ABB RobotStudio station: test1_20190225-122105.rsstn

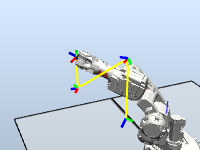
Station test1 (saved by RobotStudio 6.8.8148.134)
Layout (positions relative to the parent item):
  - IRB140_6_81_C_03_2 [mechanism, from Robots\IRB140_6_81_C_G_03.rslib] at (0, 0, 0) mm; joint values [-0.7275, 0.7441, -1.0821, -1.1758, 0.2324, 2.3516] (rad or m)
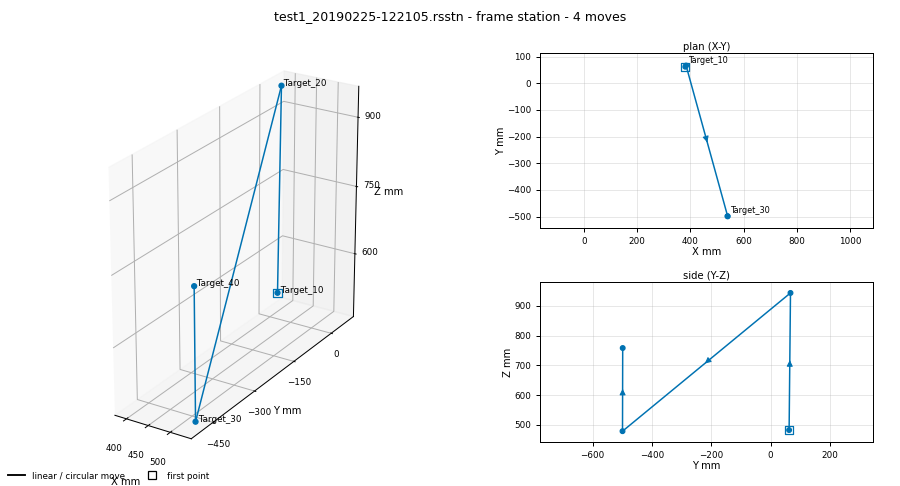
[picture p0: tool path of test1_20190225-122105.rsstn in frame station, 4 of 4 moves have a stored position in this frame; points joined in program order, loops and branches not executed]
Targets, tools, work objects and paths stored in the station, written as RAPID:
! task (no controller)
MODULE Module1
  CONST robtarget Target_10:=[[380.698967065,62.135252828,482.100752166],[0.23292276,-0.432299751,0.867192227,-0.082713687],[0,-1,-1,0],[9E+09,9E+09,9E+09,9E+09,9E+09,9E+09]];
  CONST robtarget Target_20:=[[383.520804221,66.771067435,943.970503399],[0.810617732,-0.21605232,0.523687989,-0.148226777],[0,0,-1,0],[9E+09,9E+09,9E+09,9E+09,9E+09,9E+09]];
  CONST robtarget Target_30:=[[539.642537373,-499.039538141,478.271243576],[0.556915193,0.710439618,0.428534612,0.038459103],[-1,-1,1,0],[9E+09,9E+09,9E+09,9E+09,9E+09,9E+09]];
  CONST robtarget Target_40:=[[538.902117617,-498.38021413,758.426662546],[0.778806567,0.547926937,0.283229961,0.114092908],[-1,-1,1,0],[9E+09,9E+09,9E+09,9E+09,9E+09,9E+09]];
  PROC Path_10()
    MoveL Target_10,v1000,z100,tool0\WObj:=wobj0;
    MoveL Target_20,v1000,z100,tool0\WObj:=wobj0;
    MoveL Target_30,v1000,z100,tool0\WObj:=wobj0;
    MoveL Target_40,v1000,z100,tool0\WObj:=wobj0;
  ENDPROC
ENDMODULE

